TEXTLIST CircleMode
  0 = 'Border'
  1 = 'Center'
  2 = 'Radius'
   = ''
END_TEXTLIST

(* stored: Version 1.1.0.1
   TextList CircleMode: Id {ed8b6384-2cb5-4eae-994b-8f4b848296e6} *)
